SUBAPPLICATION logiBUS_AI_Calibrate_2P_IDA_OPC (* logiBUS_AI_IDA (Analog-Eingang) mit 2-Punkt-Kalibrierung (AR_CALIBRATE_2P_REF, unabhaengig gespeicherte Rohwerte X_LOW/X_HIGH + Referenzwerte LOW_REF/HIGH_REF alle INI-persistiert) auf VT-Zahlenfelder (Rohwert + kalibrierter Wert, je eigene CNumberVariable) + Bargraph (kalibriert) + 2 VT-Tasten (CO/CS) + OPC-UA (Rohwert DWORD + kalibrierter Wert REAL, generisch, ein Kanal) *)
  (* Standard: 61499-2; Description: Copyright (c) 2026 Meisterschulen am Ostbahnhof This program and the accompanying materials are made available under the terms of the Eclipse Public License 2.0 which is available at https://www.eclipse.org/legal/epl-2.0/ SPDX-License-Identifier: EPL-2.0 *)
  (* Version 1.0, 2026-08-31, Franz Höpfinger, Meisterschulen am Ostbahnhof, initial API and implementation and/or initial documentation - Kalibrierlogik nach Vorbild Uebung_028c3_AR.SUB, aber AR_CALIBRATE_SQ (korrigierte Offset-Formel, ECC-erzwungene CO-vor-CS-Reihenfolge) statt AR_CALIBRATE *)
  (* Version 1.1, 2026-09-11, Franz Höpfinger, Meisterschulen am Ostbahnhof, Migriert auf AR_CALIBRATE_2P_REF: CO/CS speichern jetzt unabhaengig X_LOW/X_HIGH (wie AR_CALIBRATE_3P/_REF), keine ECC-erzwungene Reihenfolge mehr noetig, da CS mathematisch nie von CO abhing - nur die alte OFFSET/SCALE-Inkrementalrechnung erzwang das kuenstlich. Aeussere Schnittstelle (InputVars, VT-Tasten CO/CS, GCF-IDs) unveraendert, nur interne INI-Keys OFFSET/SCALE/ZERO/SPAN -> X_LOW/X_HIGH/LOW_REF/HIGH_REF umbenannt (Klarheit, keine bestehenden Feldgeraete betroffen). *)
  (* Version 1.2, 2026-09-17, Franz Höpfinger, Meisterschulen am Ostbahnhof, Franz: 'die Tasten vom OPC-UA Webpanel aus sollen Methoden aufrufen auf dem Steuergeraet das die Kalibrierung macht' - CO/CS bekommen einen dritten, gleichberechtigten Ausloeser: eine argumentlose OPC-UA-Methode (ID_CO_METHOD/ID_CS_METHOD, ACTION=CREATE_METHOD via SERVER_0), analog zum bereits etablierten Softkey_Aux_Method_IE-Muster (Softkey/AUX/lokale-Methode gleichberechtigt gemergt). IND->RSP-Selfloop zwingend (siehe OPC_UA_VERNETZUNG.md Punkt 12 - sonst 4s Server-Lock). Bestehende Instanzen (Ultraschall) muessen einen echten, wenn auch vorerst ungenutzten Methoden-Namen bekommen - InputVars sind nicht optional (kein WSTRING-Aequivalent zu ID_NULL). *)
  (* Version 1.3, 2026-09-17, Franz Höpfinger, Meisterschulen am Ostbahnhof, AR_CALIBRATE_2P_REF.C_LOW/C_HIGH von AX-Sockets auf reine EventInputs umgestellt (Franz: der AX-Flankenwaechter war akademisch, jeder echte Aufrufer liefert ohnehin ein atomares Event) - AX_BOOL_TO_X_CO/_CS entfallen ersatzlos, die Merge-Ketten (E_MERGE_CO_C/E_MERGE_CS_C) verbinden jetzt direkt per EventConnection mit CALIBRATE.C_LOW/C_HIGH. *)
  (* Version 1.4, 2026-09-18, Franz Höpfinger, Meisterschulen am Ostbahnhof, AX_SUBSCRIBE_CO/CS + AX_RF_TRIG_CO/CS (Toggle-Subscribe-Weiterleitung, ID_CO_READ/ID_CS_READ) ersatzlos entfernt - Cross-Station-Weiterleitung einer VT-Taste lief bisher ueber Event->Pegel(Toggle)->Event, obwohl mit ID_CO_METHOD/ID_CS_METHOD bereits ein echter Methodenaufruf existiert. Siehe OPC_UA_VERNETZUNG.md Punkt 14. E_MERGE_CO/CS schrumpfen von 4 auf 2 Quellen (lokale VT-Taste + Methode) - CO/CS-Merge-Ketten (3x E_MERGE_2 in Reihe) durch je einen einzelnen E_MERGE_2 ersetzt. *)
  (* Version 1.5, 2026-09-18, Franz Höpfinger, Meisterschulen am Ostbahnhof, Button_CO/Button_CS + METHOD_SERVER_CO/CS + E_MERGE_CO/CS (je 1x pro Taste) durch je eine Instanz des neuen wiederverwendbaren Bausteins Button_Method_IE ersetzt - identisches Muster kam 2x identisch vor, analog zu Softkey_Aux_Method_IE herausgeloest. *)
  (* Version 1.6, 2026-09-18, Franz Höpfinger, Meisterschulen am Ostbahnhof, Franz: 'kann eine SUB sein' - logiBUS_AI_IDA+AD_SPLIT_2+AD_PUBLISH_RAW+AD_TO_AUDI+AUDI_SPLIT_2+Q_NumericValue_RAW+AUDI_TO_AR durch neue SubApp logiBUS_AI_Raw_VT_AR_OPC ersetzt, AR_SPLIT_2+AR_PUBLISH_CAL+Q_NumericValue_CAL durch die bereits bestehende SubApp AR_TO_Q_Publish_OPC (dort um optionales INITO ergaenzt) - beide Muster kamen identisch auch in logiBUS_AI_Calibrate_3P_IDA_OPC vor. *)
  (* Version 1.7, 2026-09-20, Franz Höpfinger, Meisterschulen am Ostbahnhof, Rohwert-Anzeige an den Kalibrierpunkten (Zero-Raw/Span-Raw) ergaenzt, Franz: 'im Web-Panel und im IOP die Roh-Werte mit anzeigen'. CALIBRATE.X_LOW/X_HIGH (AR2, bisher nur an INI_X_LOW/INI_X_HIGH angeschlossen) werden ueber neue TapZeroRaw/TapSpanRaw (MyLib::sys::AR2_TAP_TO_AR) abgezapft, ohne die bestehende Persistenz-/Restore-Kette zu aendern, und ueber neue PublishZeroRaw/PublishSpanRaw (MyLib::sys::AR_TO_Q_Publish_OPC) als reine Nur-Lese-Anzeige (VT CNumberVariable + OPC-UA Publish) exponiert. Neue InputVars stObjZeroRaw/stObjSpanRaw (VT-Objekt) + ID_ZERO_RAW_WRITE/ID_SPAN_RAW_WRITE (OPC-UA-Adresse). *)
  (* Version 1.9, 2026-09-21, Franz Höpfinger, Meisterschulen am Ostbahnhof, Code-Review-Fund (PR #260): INI_X_HIGH.DEFAULT_VALUE stand auf REAL#1.0 statt 0.0 - AR_CALIBRATE_2P_REF's neuer xHighCal-Kalibriert-Flag (v1.3, prueft X_HIGH.DI1 <> 0.0) latchte dadurch bei JEDEM Boot sofort TRUE, obwohl HIGH nie kalibriert wurde (fabricated reference statt Partial-Kalibrierung-Fallback). Default auf REAL#0.0 korrigiert, passend zu INI_X_LOW und zum Flag-Vergleich. *)
  (* Version 1.8, 2026-09-21, Franz Höpfinger, Meisterschulen am Ostbahnhof, AR_CALIBRATE_2P_REF hat jetzt ein INIT/QI/QO-Enable-Pattern (genauso wie AR_CALIBRATE_3P_REF: Bugfix Garbage-Interpolation bei nur einem kalibrierten Punkt + xClipping) - CALIBRATE bekommt Parameter QI=TRUE (wie die INI_X_LOW/X_HIGH-Instanzen), sonst bleibt die FB im START-Zustand haengen und REQ laeuft nie. *)
  (* Version 1.10, 2026-09-23, Franz Hoepfinger, Meisterschulen am Ostbahnhof, INI_LOW_REF.DEFAULT_VALUE/INI_HIGH_REF.DEFAULT_VALUE waren fest verdrahtet (0.0/100.0) - neue InputVars rLowRefDefault/rHighRefDefault machen die Erstinbetriebnahme-Referenzwerte pro Instanz konfigurierbar (Druck braucht 250.0 statt Fuellbands 100.0), bestehende Instanzen unveraendert per Default. *)
  (* Version 1.11, 2026-09-27, Franz Höpfinger, Meisterschulen am Ostbahnhof, Neuer Plug CAL_OUT (kalibrierter Wert, lokal AR) - bisher verliess der kalibrierte Wert diesen Typ nur per OPC-UA-Publish, was fuer lokale Weiterverarbeitung auf einer VT-losen Station (z.B. Fuellband-oben-Schwellwert) einen unnoetigen Remote-Roundtrip erzwang. CALIBRATE.Y jetzt per neuem AR_SPLIT_2 auf PublishCal UND CAL_OUT verzweigt (Fan-out-Regel: nie direkt). *)
  PACKAGE MyLib::sys;
  IMPORT isobus::UT::Q::const::IDs::ID_NULL;
  IMPORT logiBUS::io::AI::logiBUS_AI;
  IMPORT logiBUS::io::AI::logiBUS_AI_S;
  IMPORT logiBUS::utils::conversion::phys::NumericObjectPool_S;
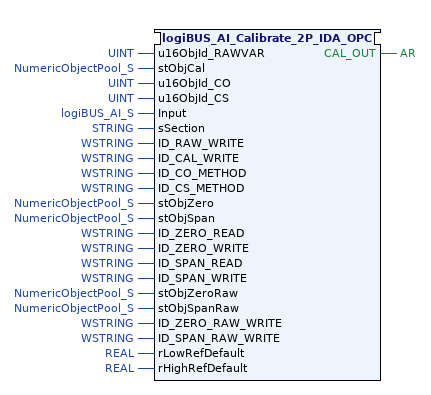
  VAR_INPUT
    u16ObjId_RAWVAR : UINT := ID_NULL; (* Object ID CNumberVariable (Rohwert 0-4095, unkalibriert, reine Diagnose-Anzeige) *)
    stObjCal : logiBUS::utils::conversion::phys::NumericObjectPool_S := (u16ObjId := ID_NULL, r32Scale := 1.0, i32Offset := 0, u8Decimals := 1); (* Object ID + Scale/Offset/Decimals CNumberVariable (kalibrierter Wert, eigene, unabhaengige CNumberVariable) *)
    u16ObjId_CO : UINT := ID_NULL; (* Object ID Taste 'CO' (Kalibrier-Nullpunkt: Referenz 1 anlegen, dann druecken) *)
    u16ObjId_CS : UINT := ID_NULL; (* Object ID Taste 'CS' (Kalibrier-Spanne: Referenz 2 anlegen, dann druecken - erst nach CO moeglich) *)
    Input : logiBUS::io::AI::logiBUS_AI_S := logiBUS_AI::Invalid; (* Identify the Input AnalogInput_I1..I8 *)
    sSection : STRING; (* INI-Sektionsname fuer OFFSET/SCALE-Persistenz - pro Kanal eindeutig (z.B. 'AI_Calibrate_I1'), sonst kollidieren die Kanaele in settings.ini *)
    ID_RAW_WRITE : WSTRING; (* Rohwert-Ruckmelde-Adresse (DWORD 0-4095, ACTION=PUBLISH) *)
    ID_CAL_WRITE : WSTRING; (* Kalibrierter-Wert-Ruckmelde-Adresse (REAL, ACTION=PUBLISH) *)
    ID_CO_METHOD : WSTRING; (* Methodenadresse (ACTION=CREATE_METHOD) fuer den argumentlosen CO-Trigger - gleichberechtigt zur lokalen VT-Taste aufrufbar, sowohl vom OPC-UA-Dashboard als auch per CLIENT_0 von einer anderen Station (Cross-Station-Weiterleitung einer dortigen VT-Taste, siehe OPC_UA_VERNETZUNG.md Punkt 14 - kein Toggle/Subscribe-Umweg mehr) *)
    ID_CS_METHOD : WSTRING; (* Methodenadresse (ACTION=CREATE_METHOD) fuer den argumentlosen CS-Trigger - siehe ID_CO_METHOD *)
    stObjZero : logiBUS::utils::conversion::phys::NumericObjectPool_S := (u16ObjId := ID_NULL, r32Scale := 1.0, i32Offset := 0, u8Decimals := 1); (* Object ID + Scale/Offset/Decimals CNumberVariable (ZERO-Referenzwert, VT-Eingabefeld + OPC-UA) *)
    stObjSpan : logiBUS::utils::conversion::phys::NumericObjectPool_S := (u16ObjId := ID_NULL, r32Scale := 1.0, i32Offset := 0, u8Decimals := 1); (* Object ID + Scale/Offset/Decimals CNumberVariable (SPAN-Referenzwert, VT-Eingabefeld + OPC-UA) *)
    ID_ZERO_READ : WSTRING; (* Remote-Subscribe-Adresse ZERO-Referenzwert (REAL, ACTION=SUBSCRIBE) *)
    ID_ZERO_WRITE : WSTRING; (* Remote-Echo-Adresse ZERO-Referenzwert (REAL, ACTION=PUBLISH) *)
    ID_SPAN_READ : WSTRING; (* Remote-Subscribe-Adresse SPAN-Referenzwert (REAL, ACTION=SUBSCRIBE) *)
    ID_SPAN_WRITE : WSTRING; (* Remote-Echo-Adresse SPAN-Referenzwert (REAL, ACTION=PUBLISH) *)
    stObjZeroRaw : logiBUS::utils::conversion::phys::NumericObjectPool_S := (u16ObjId := ID_NULL, r32Scale := 1.0, i32Offset := 0, u8Decimals := 1); (* Object ID + Scale/Offset/Decimals CNumberVariable (Rohwert am ZERO-Kalibrierpunkt, reine Diagnose-Anzeige) *)
    stObjSpanRaw : logiBUS::utils::conversion::phys::NumericObjectPool_S := (u16ObjId := ID_NULL, r32Scale := 1.0, i32Offset := 0, u8Decimals := 1); (* Object ID + Scale/Offset/Decimals CNumberVariable (Rohwert am SPAN-Kalibrierpunkt, reine Diagnose-Anzeige) *)
    ID_ZERO_RAW_WRITE : WSTRING; (* Rohwert-am-ZERO-Kalibrierpunkt-Publish-Adresse (REAL, ACTION=PUBLISH) *)
    ID_SPAN_RAW_WRITE : WSTRING; (* Rohwert-am-SPAN-Kalibrierpunkt-Publish-Adresse (REAL, ACTION=PUBLISH) *)
    rLowRefDefault : REAL := REAL#0.0; (* Erstinbetriebnahme-Standardwert LOW_REF (INI_LOW_REF.DEFAULT_VALUE), bevor der Bediener selbst kalibriert - Fuellband/die meisten Sensoren: 0.0 *)
    rHighRefDefault : REAL := REAL#100.0; (* Erstinbetriebnahme-Standardwert HIGH_REF (INI_HIGH_REF.DEFAULT_VALUE), bevor der Bediener selbst kalibriert - z.B. 250.0 fuer Druck (0-250bar), 100.0 fuer Fuellband-Winkel (Prozent) *)
  END_VAR
  PLUGS
    CAL_OUT : adapter::types::unidirectional::AR; (* Kalibrierter Wert, lokal (= CALIBRATE.Y) - fuer Weiterverarbeitung auf derselben Station ohne OPC-UA-Roundtrip *)
  END_PLUGS
  FBS
    CALIBRATE : adapter::Engineering::measurements::AR_CALIBRATE_2P_REF(QI := TRUE, xClipping := FALSE);
    INI_X_LOW : eclipse4diac::storage::INI_AR2(QI := TRUE, SETM := TRUE, KEY := 'X_LOW', DEFAULT_VALUE := REAL#0.0);
    INI_X_HIGH : eclipse4diac::storage::INI_AR2(QI := TRUE, SETM := TRUE, KEY := 'X_HIGH', DEFAULT_VALUE := REAL#0.0);
    INI_LOW_REF : eclipse4diac::storage::INI_AR2(QI := TRUE, SETM := TRUE, KEY := 'LOW_REF');
    INI_HIGH_REF : eclipse4diac::storage::INI_AR2(QI := TRUE, SETM := TRUE, KEY := 'HIGH_REF');
    TapZeroRaw : adapter::events::bidirectional::AR2_SPLIT_FWD_REV;
    TapSpanRaw : adapter::events::bidirectional::AR2_SPLIT_FWD_REV;
    AR_SPLIT_2_Cal : adapter::events::unidirectional::AR_SPLIT_2;
  END_FBS
  SUBAPPS
    InputRaw : MyLib::sys::logiBUS_AI_Raw_VT_AR_OPC;
    Y_OFFSET_LIT : MyLib::sys::NumericValue_TO_AR2_OPC;
    Y_SCALE_LIT : MyLib::sys::NumericValue_TO_AR2_OPC;
    TriggerCO : MyLib::sys::Button_Method_IE;
    TriggerCS : MyLib::sys::Button_Method_IE;
    PublishCal : MyLib::sys::AR_TO_Q_Publish_OPC;
    PublishZeroRaw : MyLib::sys::AR_TO_Q_Publish_OPC;
    PublishSpanRaw : MyLib::sys::AR_TO_Q_Publish_OPC;
  END_SUBAPPS
  EVENT_CONNECTIONS
    TriggerCO.IND TO CALIBRATE.C_LOW;
    TriggerCS.IND TO CALIBRATE.C_HIGH;
  END_CONNECTIONS
  DATA_CONNECTIONS
    Input TO InputRaw.Input;
    u16ObjId_RAWVAR TO InputRaw.u16ObjId_RAWVAR;
    stObjCal TO PublishCal.stObj;
    u16ObjId_CO TO TriggerCO.u16ObjId;
    u16ObjId_CS TO TriggerCS.u16ObjId;
    sSection TO INI_X_LOW.SECTION;
    sSection TO INI_X_HIGH.SECTION;
    sSection TO INI_LOW_REF.SECTION;
    sSection TO INI_HIGH_REF.SECTION;
    rLowRefDefault TO INI_LOW_REF.DEFAULT_VALUE;
    rHighRefDefault TO INI_HIGH_REF.DEFAULT_VALUE;
    ID_RAW_WRITE TO InputRaw.ID_RAW_WRITE;
    ID_CAL_WRITE TO PublishCal.ID_WRITE;
    ID_CO_METHOD TO TriggerCO.ID_METHOD;
    ID_CS_METHOD TO TriggerCS.ID_METHOD;
    stObjZero TO Y_OFFSET_LIT.stObj;
    ID_ZERO_READ TO Y_OFFSET_LIT.ID_READ;
    ID_ZERO_WRITE TO Y_OFFSET_LIT.ID_WRITE;
    stObjSpan TO Y_SCALE_LIT.stObj;
    ID_SPAN_READ TO Y_SCALE_LIT.ID_READ;
    ID_SPAN_WRITE TO Y_SCALE_LIT.ID_WRITE;
    stObjZeroRaw TO PublishZeroRaw.stObj;
    ID_ZERO_RAW_WRITE TO PublishZeroRaw.ID_WRITE;
    stObjSpanRaw TO PublishSpanRaw.stObj;
    ID_SPAN_RAW_WRITE TO PublishSpanRaw.ID_WRITE;
  END_CONNECTIONS
  ADAPTER_CONNECTIONS
    InputRaw.AR_OUT TO CALIBRATE.X;
    CALIBRATE.X_LOW TO TapZeroRaw.IN;
    TapZeroRaw.OUT TO INI_X_LOW.VAL;
    TapZeroRaw.REV_OUT TO PublishZeroRaw.AR_IN;
    CALIBRATE.X_HIGH TO TapSpanRaw.IN;
    TapSpanRaw.OUT TO INI_X_HIGH.VAL;
    TapSpanRaw.REV_OUT TO PublishSpanRaw.AR_IN;
    CALIBRATE.LOW_REF TO INI_LOW_REF.VAL;
    CALIBRATE.HIGH_REF TO INI_HIGH_REF.VAL;
    Y_OFFSET_LIT.VALUEO TO CALIBRATE.Y_LOW;
    Y_SCALE_LIT.VALUEO TO CALIBRATE.Y_HIGH;
    CALIBRATE.Y TO AR_SPLIT_2_Cal.IN;
    AR_SPLIT_2_Cal.OUT1 TO PublishCal.AR_IN;
    AR_SPLIT_2_Cal.OUT2 TO CAL_OUT;
  END_CONNECTIONS
END_SUBAPPLICATION
